PROGRAM ControlElvSFC
VAR
	SendDequeue: INT;
	ResetDequeue: BOOL;
	SendDequeue1: BOOL;
	Reset: INT;
	ResetDequeue_1: BOOL;
	SendDequeue2: BOOL;
	ResetDequeue_2: BOOL;
	SendDequeue3: BOOL;
	ResetDequeue_3: BOOL;
END_VAR

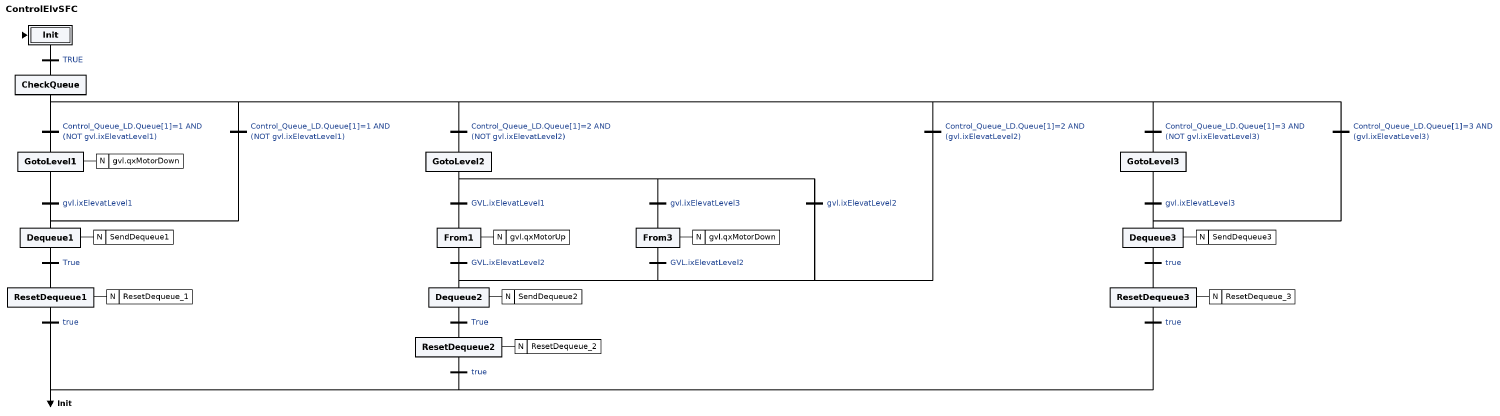
INITIAL_STEP Init:
END_STEP
TRANSITION FROM Init TO CheckQueue
    := TRUE;
END_TRANSITION
STEP CheckQueue:
END_STEP
TRANSITION FROM CheckQueue TO GotoLevel1
    := Control_Queue_LD.Queue[1]=1 AND (NOT gvl.ixElevatLevel1);
END_TRANSITION
STEP GotoLevel1:
    gvl.qxMotorDown(N);
END_STEP
TRANSITION FROM GotoLevel1 TO Dequeue1
    := gvl.ixElevatLevel1;
END_TRANSITION
TRANSITION FROM CheckQueue TO Dequeue1
    := Control_Queue_LD.Queue[1]=1 AND (NOT gvl.ixElevatLevel1);
END_TRANSITION
STEP Dequeue1:
    SendDequeue1(N);
END_STEP
TRANSITION FROM Dequeue1 TO ResetDequeue1
    := True;
END_TRANSITION
STEP ResetDequeue1:
    ResetDequeue_1(N);
END_STEP
TRANSITION FROM ResetDequeue1 TO Init
    := true;
END_TRANSITION
TRANSITION FROM CheckQueue TO GotoLevel2
    := Control_Queue_LD.Queue[1]=2 AND (NOT gvl.ixElevatLevel2);
END_TRANSITION
STEP GotoLevel2:
END_STEP
TRANSITION FROM GotoLevel2 TO From1
    := GVL.ixElevatLevel1;
END_TRANSITION
STEP From1:
    gvl.qxMotorUp(N);
END_STEP
TRANSITION FROM From1 TO Dequeue2
    := GVL.ixElevatLevel2;
END_TRANSITION
TRANSITION FROM GotoLevel2 TO From3
    := gvl.ixElevatLevel3;
END_TRANSITION
STEP From3:
    gvl.qxMotorDown(N);
END_STEP
TRANSITION FROM From3 TO Dequeue2
    := GVL.ixElevatLevel2;
END_TRANSITION
TRANSITION FROM GotoLevel2 TO Dequeue2
    := gvl.ixElevatLevel2;
END_TRANSITION
TRANSITION FROM CheckQueue TO Dequeue2
    := Control_Queue_LD.Queue[1]=2 AND (gvl.ixElevatLevel2);
END_TRANSITION
STEP Dequeue2:
    SendDequeue2(N);
END_STEP
TRANSITION FROM Dequeue2 TO ResetDequeue2
    := True;
END_TRANSITION
STEP ResetDequeue2:
    ResetDequeue_2(N);
END_STEP
TRANSITION FROM ResetDequeue2 TO Init
    := true;
END_TRANSITION
TRANSITION FROM CheckQueue TO GotoLevel3
    := Control_Queue_LD.Queue[1]=3 AND (NOT gvl.ixElevatLevel3);
END_TRANSITION
STEP GotoLevel3:
END_STEP
TRANSITION FROM GotoLevel3 TO Dequeue3
    := gvl.ixElevatLevel3;
END_TRANSITION
TRANSITION FROM CheckQueue TO Dequeue3
    := Control_Queue_LD.Queue[1]=3 AND (gvl.ixElevatLevel3);
END_TRANSITION
STEP Dequeue3:
    SendDequeue3(N);
END_STEP
TRANSITION FROM Dequeue3 TO ResetDequeue3
    := true;
END_TRANSITION
STEP ResetDequeue3:
    ResetDequeue_3(N);
END_STEP
TRANSITION FROM ResetDequeue3 TO Init
    := true;
END_TRANSITION

END_PROGRAM

(* stored: Version 1.1.0.1, ProductVersion 3.1.4024.12
   POU ControlElvSFC: Id {7824d25e-4d76-4290-ade9-26c4a0b6feeb}, SpecialFunc None *)
